(* IEC 61131-3 sources: std_i2980_v2.06_cp053/Source/IMM/ieccontrol/NozzleGeneral, 10 files *)

(* ---- ABButtonControl.pu ---- *)
IMPORT_OVER_LISTFILE
 IS_LINKED
, cBarInvert
, tyPanelButton
, tevPanelButtonRegisterData
, tevPanelButtonRegister
, ABManualButton
, tsDeviceId
, tsPanelButton

END_IMPORT

ALGORITHM_BLOCK ABButtonControl #DUMMY_EDIT_BLOCK

SYSTEM_VAR
 sv_bInitStart : BOOL;
 sv_bDeviceReady : BOOL;
 sv_bTransducerAvailable : BOOL;
 sv_iPanelMovementSelector : DINT;
 sv_PanelButtons : tyPanelButton;
 di_ButtonFwd : BOOL;
 di_ButtonBwd : BOOL;
 sv_bNozzleFwd : BOOL;
 sv_bNozzleBwd : BOOL;
 sv_bButtonFwd : BOOL;
 sv_bButtonBwd : BOOL;
 di_ButtonGeneral1 : BOOL;
 di_ButtonGeneral2 : BOOL;
 sv_DeviceId : tsDeviceId;
 sv_rNozzlePosition : REAL;
 sv_rNozzleStroke : REAL;
END_VAR

SYSTEM_OBJECT
 evPanelButtonRegister : tevPanelButtonRegister;
 PU_Task_7 : TASK;
 PU_Task_13 : TASK;
END_OBJECT

VAR
 evPanelButtonRegisterData : tevPanelButtonRegisterData;
 abManualButton : ABManualButton;
 mpbButtonGeneralFwd : REFTO BOOL;
 mpbButtonGeneralBwd : REFTO BOOL;
 mbDIButtonFwdLinked : BOOL;
 mbDIButtonBwdLinked : BOOL;
 mbDIButtonGeneralFwdLinked : BOOL;
 mbDIButtonGeneralBwdLinked : BOOL;
 mpiPanelMovementSelector : REFTO DINT;
END_VAR

VAR CONSTANT
 cButtonMoveFwdBwd : DINT := 1;
END_VAR

POSTUPDATE_ALGORITHM pRegisterButtons ON PU_Task_13 WITH sv_bInitStart

#BEGIN_EDIT_BLOCK
(**************************************** WARNING ********************************************
 *** The KEBA Kemro K2 System including software is not intended for safety control tasks! ***
 ***                       For further information see Comment tab!                        ***
 *********************************************************************************************)

mpbButtonGeneralFwd := EMPTY;
mpbButtonGeneralBwd := EMPTY;

mbDIButtonFwdLinked := IS_LINKED(di_ButtonFwd);
mbDIButtonBwdLinked := IS_LINKED(di_ButtonBwd);

mbDIButtonGeneralFwdLinked := IS_LINKED(di_ButtonGeneral1);
mbDIButtonGeneralBwdLinked := IS_LINKED(di_ButtonGeneral2);

IF (mbDIButtonGeneralFwdLinked AND mbDIButtonGeneralBwdLinked) THEN
    mpiPanelMovementSelector := @sv_iPanelMovementSelector;
END_IF;

evPanelButtonRegisterData.Button.nPanelButtonType := nPanelButtonMovement;
evPanelButtonRegisterData.Button.iCompId := sv_DeviceId.CompId;
evPanelButtonRegisterData.Button.iIndexId := sv_DeviceId.IndexId;
evPanelButtonRegisterData.Button.iButtonId := cButtonMoveFwdBwd;
evPanelButtonRegisterData.Button.pbActionVar1 := @sv_bButtonFwd;
evPanelButtonRegisterData.Button.pbActionVar2 := @sv_bButtonBwd;
IF sv_bTransducerAvailable THEN
   evPanelButtonRegisterData.Button.Optional.prActVar := @sv_rNozzlePosition;
END_IF;
evPanelButtonRegisterData.Button.Optional.prMaxVar := @sv_rNozzleStroke;
evPanelButtonRegisterData.Button.Optional.prMinVar :=  EMPTY;
evPanelButtonRegisterData.Button.Optional.iBarAttr := cBarInvert;
evPanelButtonRegisterData.Button.Optional.pbLimitSwitch1 := @sv_bNozzleFwd;
evPanelButtonRegisterData.Button.Optional.pbLimitSwitch2 := @sv_bNozzleBwd;
SET_EVENT(evPanelButtonRegister, evPanelButtonRegisterData);

;#END_EDIT_BLOCK END_ALGORITHM

POSTUPDATE_ALGORITHM pButtonFwd ON PU_Task_7 WITH di_ButtonFwd, sv_bButtonFwd, mpbButtonGeneralFwd^

VAR
 bButton : BOOL;
END_VAR
#BEGIN_EDIT_BLOCK
(**************************************** WARNING ********************************************
 *** The KEBA Kemro K2 System including software is not intended for safety control tasks! ***
 ***                       For further information see Comment tab!                        ***
 *********************************************************************************************)

// soft panel button
bButton := sv_bButtonFwd;

// hw panel button
IF mbDIButtonFwdLinked THEN
    bButton := bButton OR di_ButtonFwd;
END_IF;

// external panel button
IF CHECK_REF(mpbButtonGeneralFwd^) THEN
    bButton := bButton OR mpbButtonGeneralFwd^;
END_IF;

abManualButton.aButtonFwd(bButtonFwd := bButton);

;#END_EDIT_BLOCK END_ALGORITHM

POSTUPDATE_ALGORITHM pButtonBwd ON PU_Task_7 WITH di_ButtonBwd, sv_bButtonBwd, mpbButtonGeneralBwd^

VAR
 bButton : BOOL;
END_VAR
#BEGIN_EDIT_BLOCK
(**************************************** WARNING ********************************************
 *** The KEBA Kemro K2 System including software is not intended for safety control tasks! ***
 ***                       For further information see Comment tab!                        ***
 *********************************************************************************************)

// soft panel button
bButton := sv_bButtonBwd;

// hw panel button
IF mbDIButtonBwdLinked THEN
    bButton := bButton OR di_ButtonBwd;
END_IF;

// external panel button
IF CHECK_REF(mpbButtonGeneralBwd^) THEN
    bButton := bButton OR mpbButtonGeneralBwd^;
END_IF;

abManualButton.aButtonBwd(bButtonBwd := bButton);

;#END_EDIT_BLOCK END_ALGORITHM

POSTUPDATE_ALGORITHM pMoveSelectorChanged ON PU_Task_7 WITH mpiPanelMovementSelector^

VAR
 Button : tsPanelButton;
END_VAR
#BEGIN_EDIT_BLOCK
(**************************************** WARNING ********************************************
 *** The KEBA Kemro K2 System including software is not intended for safety control tasks! ***
 ***                       For further information see Comment tab!                        ***
 *********************************************************************************************)

mpbButtonGeneralFwd := EMPTY;
mpbButtonGeneralBwd := EMPTY;

IF (NOT sv_bDeviceReady) THEN
    // stop active movements
    abManualButton.aButtonBwd(bButtonBwd := FALSE);
    abManualButton.aButtonFwd(bButtonFwd := FALSE);
END_IF;

IF (sv_iPanelMovementSelector > 0) THEN
    Button := sv_PanelButtons[sv_iPanelMovementSelector];
    IF Button.iCompId = sv_DeviceId.CompId AND
        Button.iIndexId = sv_DeviceId.IndexId THEN
        IF Button.iButtonId = cButtonMoveFwdBwd THEN
            mpbButtonGeneralFwd := @di_ButtonGeneral1;
            mpbButtonGeneralBwd := @di_ButtonGeneral2;
        END_IF;
    END_IF;
END_IF;

;#END_EDIT_BLOCK END_ALGORITHM

END_ALGORITHM_BLOCK

#END_OF_IEC_PART

@Puma @IecEditor 6 150 @Pou 25
@@@BEG_Comment@@@

@@@END_Comment@@@

@BEG_Contents

@BEG_Func
@RT(17)FuncTreeContainer
1
@Var @RT(9)IS_LINKED @RT(0) @T @T @DERIVED 0 @F @RT(22)KEBA_STANDARD_FUNCTION @F
@T
@BEG_Attrib
0 @RT(0) @RT(0)
@END_Attrib
1 1 @F @F @F @F

@END_Func

@BEG_Const
@RT(18)ConstTreeContainer
1
@Var @RT(10)cBarInvert @RT(0) @T @F @DT @RT(4)BYTE @RT(0) @T @T @BASIC 0 @F
@F @F
@T
@BEG_Attrib
0 @RT(1)1 @RT(0)
@END_Attrib
1 1 @F @F @F @F

@END_Const

@BEG_Export

@BEG_Kind
@ALGORITHM_BLOCK @RT(15)ABButtonControl @STRUCTURED_TEXT
@RT(0) @RT(0) @RT(0)
@END_Kind

@BEG_Dcl
@RT(16)DclTreeContainer
29
@Var @RT(13)sv_bInitStart @RT(0) @T @T @RENAMED 0 @T @T @DT @RT(4)BOOL @RT(0) @T @T @BASIC 0 @F
@F @F
@T
@BEG_Attrib
3 @RT(0) @RT(0) @RT(0)
@END_Attrib
1 8 @F @F @F @F

@Var @RT(15)sv_bDeviceReady @RT(0) @T @T @RENAMED 0 @T @T @DT @RT(4)BOOL @RT(0) @T @T @BASIC 0 @F
@F @F
@T
@BEG_Attrib
3 @RT(0) @RT(0) @RT(0)
@END_Attrib
1 8 @F @F @F @F

@Var @RT(23)sv_bTransducerAvailable @RT(0) @T @F @DT @RT(4)BOOL @RT(0) @T @T @BASIC 0 @F
@F @F
@T
@BEG_Attrib
3 @RT(0) @RT(0) @RT(0)
@END_Attrib
1 8 @F @F @F @F

@Var @RT(25)sv_iPanelMovementSelector @RT(0) @T @F @DT @RT(4)DINT @RT(0) @T @T @BASIC 0 @F
@F @F
@T
@BEG_Attrib
3 @RT(0) @RT(0) @RT(0)
@END_Attrib
1 8 @F @F @F @F

@Var @RT(15)sv_PanelButtons @RT(0) @T @T @DERIVED 0 @T @T @DT @RT(13)tyPanelButton @RT(0) @T @T @UNKNOWN 0 @F
@F @F
@T
@BEG_Attrib
3 @RT(0) @RT(0) @RT(0)
@END_Attrib
1 8 @F @F @F @F

@Var @RT(25)evPanelButtonRegisterData @RT(0) @T @T @DERIVED 0 @T @T @DT @RT(26)tevPanelButtonRegisterData @RT(0) @T @T @UNKNOWN 0 @F
@F @F
@T
@BEG_Attrib
3 @RT(0) @RT(0) @RT(0)
@END_Attrib
1 0 @F @F @F @F

@Var @RT(21)evPanelButtonRegister @RT(0) @T @T @DERIVED 0 @T @T @DT @RT(22)tevPanelButtonRegister @RT(0) @T @T @UNKNOWN 0 @F
@F @F
@T
@BEG_Attrib
3 @RT(0) @RT(0) @RT(0)
@END_Attrib
1 7 @F @F @F @F

@Var @RT(14)abManualButton @RT(0) @T @T @DERIVED 0 @T @T @DT @RT(14)ABManualButton @RT(0) @T @T @UNKNOWN 0 @F
@F @F
@T
@BEG_Attrib
3 @RT(0) @RT(0) @RT(0)
@END_Attrib
1 0 @F @F @F @F

@Var @RT(12)di_ButtonFwd @RT(0) @T @T @RENAMED 0 @T @T @DT @RT(4)BOOL @RT(0) @T @T @BASIC 0 @F
@F @F
@T
@BEG_Attrib
3 @RT(0) @RT(0) @RT(0)
@END_Attrib
1 8 @F @F @F @F

@Var @RT(12)di_ButtonBwd @RT(0) @T @T @RENAMED 0 @T @T @DT @RT(4)BOOL @RT(0) @T @T @BASIC 0 @F
@F @F
@T
@BEG_Attrib
3 @RT(0) @RT(0) @RT(0)
@END_Attrib
1 8 @F @F @F @F

@Var @RT(13)sv_bNozzleFwd @RT(0) @T @T @RENAMED 0 @T @T @DT @RT(4)BOOL @RT(0) @T @T @BASIC 0 @F
@F @F
@T
@BEG_Attrib
3 @RT(0) @RT(0) @RT(0)
@END_Attrib
1 8 @F @F @F @F

@Var @RT(13)sv_bNozzleBwd @RT(0) @T @T @RENAMED 0 @T @T @DT @RT(4)BOOL @RT(0) @T @T @BASIC 0 @F
@F @F
@T
@BEG_Attrib
3 @RT(0) @RT(0) @RT(0)
@END_Attrib
1 8 @F @F @F @F

@Var @RT(13)sv_bButtonFwd @RT(0) @T @T @RENAMED 0 @T @T @DT @RT(4)BOOL @RT(0) @T @T @BASIC 0 @F
@F @F
@T
@BEG_Attrib
3 @RT(0) @RT(0) @RT(0)
@END_Attrib
1 8 @F @F @F @F

@Var @RT(13)sv_bButtonBwd @RT(0) @T @T @RENAMED 0 @T @T @DT @RT(4)BOOL @RT(0) @T @T @BASIC 0 @F
@F @F
@T
@BEG_Attrib
3 @RT(0) @RT(0) @RT(0)
@END_Attrib
1 8 @F @F @F @F

@Var @RT(17)di_ButtonGeneral1 @RT(0) @T @F @DT @RT(4)BOOL @RT(0) @T @T @BASIC 0 @F
@F @F
@T
@BEG_Attrib
3 @RT(0) @RT(0) @RT(0)
@END_Attrib
1 8 @F @F @F @F

@Var @RT(17)di_ButtonGeneral2 @RT(0) @T @F @DT @RT(4)BOOL @RT(0) @T @T @BASIC 0 @F
@F @F
@T
@BEG_Attrib
3 @RT(0) @RT(0) @RT(0)
@END_Attrib
1 8 @F @F @F @F

@Var @RT(9)PU_Task_7 @RT(0) @T @F @DT @RT(4)TASK @RT(0) @T @T @BASIC 0 @F
@F @F
@T
@BEG_Attrib
3 @RT(0) @RT(0) @RT(0)
@END_Attrib
1 7 @F @F @F @F

@Var @RT(10)PU_Task_13 @RT(0) @T @T @RENAMED 0 @T @T @DT @RT(4)TASK @RT(0) @T @T @BASIC 0 @F
@F @F
@T
@BEG_Attrib
3 @RT(0) @RT(0) @RT(0)
@END_Attrib
1 7 @F @F @F @F

@Var @RT(11)sv_DeviceId @RT(0) @T @T @DERIVED 0 @T @T @DT @RT(10)tsDeviceId @RT(0) @T @T @UNKNOWN 0 @F
@F @F
@T
@BEG_Attrib
3 @RT(0) @RT(0) @RT(0)
@END_Attrib
1 8 @F @F @F @F

@Var @RT(18)sv_rNozzlePosition @RT(0) @T @F @DT @RT(4)REAL @RT(0) @T @T @BASIC 0 @F
@F @F
@T
@BEG_Attrib
3 @RT(0) @RT(0) @RT(0)
@END_Attrib
1 8 @F @F @F @F

@Var @RT(16)sv_rNozzleStroke @RT(0) @T @F @DT @RT(4)REAL @RT(0) @T @T @BASIC 0 @F
@F @F
@T
@BEG_Attrib
3 @RT(0) @RT(0) @RT(0)
@END_Attrib
1 8 @F @F @F @F

@Var @RT(17)cButtonMoveFwdBwd @RT(0) @T @F @DT @RT(4)DINT @RT(0) @T @T @BASIC 0 @F
@F @F
@T
@BEG_Attrib
3 @RT(1)1 @RT(0) @RT(0)
@END_Attrib
1 15 @F @F @F @F

@Var @RT(19)mpbButtonGeneralFwd @RT(0) @T @T @REFTO 0 @T @DT @RT(4)BOOL @RT(0) @T @T @BASIC 0 @F
@F @F
@T
@BEG_Attrib
3 @RT(0) @RT(0) @RT(0)
@END_Attrib
1 0 @F @F @F @F

@Var @RT(19)mpbButtonGeneralBwd @RT(0) @T @T @REFTO 0 @T @DT @RT(4)BOOL @RT(0) @T @T @BASIC 0 @F
@F @F
@T
@BEG_Attrib
3 @RT(0) @RT(0) @RT(0)
@END_Attrib
1 0 @F @F @F @F

@Var @RT(19)mbDIButtonFwdLinked @RT(0) @T @F @DT @RT(4)BOOL @RT(0) @T @T @BASIC 0 @F
@F @F
@T
@BEG_Attrib
3 @RT(0) @RT(0) @RT(0)
@END_Attrib
1 0 @F @F @F @F

@Var @RT(19)mbDIButtonBwdLinked @RT(0) @T @F @DT @RT(4)BOOL @RT(0) @T @T @BASIC 0 @F
@F @F
@T
@BEG_Attrib
3 @RT(0) @RT(0) @RT(0)
@END_Attrib
1 0 @F @F @F @F

@Var @RT(26)mbDIButtonGeneralFwdLinked @RT(0) @T @F @DT @RT(4)BOOL @RT(0) @T @T @BASIC 0 @F
@F @F
@T
@BEG_Attrib
3 @RT(0) @RT(0) @RT(0)
@END_Attrib
1 0 @F @F @F @F

@Var @RT(26)mbDIButtonGeneralBwdLinked @RT(0) @T @F @DT @RT(4)BOOL @RT(0) @T @T @BASIC 0 @F
@F @F
@T
@BEG_Attrib
3 @RT(0) @RT(0) @RT(0)
@END_Attrib
1 0 @F @F @F @F

@Var @RT(24)mpiPanelMovementSelector @RT(0) @T @T @REFTO 0 @T @DT @RT(4)DINT @RT(0) @T @T @BASIC 0 @F
@F @F
@T
@BEG_Attrib
3 @RT(0) @RT(0) @RT(0)
@END_Attrib
1 0 @F @F @F @F

@END_Dcl

@END_Export

@BEG_Body

4

@BEG_Export

@BEG_Algo
@POSTUPDATE_ALGORITHM @RT(16)pRegisterButtons @STRUCTURED_TEXT
@RT(0) @RT(13)sv_bInitStart @RT(10)PU_Task_13 @F @F
@END_Algo

@BEG_Dcl
@RT(16)DclTreeContainer
0
@END_Dcl

@END_Export

@BEG_Export

@BEG_Algo
@POSTUPDATE_ALGORITHM @RT(10)pButtonFwd @STRUCTURED_TEXT
@RT(0) @RT(49)di_ButtonFwd, sv_bButtonFwd, mpbButtonGeneralFwd^ @RT(9)PU_Task_7 @F @F
@END_Algo

@BEG_Dcl
@RT(16)DclTreeContainer
1
@Var @RT(7)bButton @RT(0) @T @F @DT @RT(4)BOOL @RT(0) @T @T @BASIC 0 @F
@F @F
@T
@BEG_Attrib
3 @RT(0) @RT(0) @RT(0)
@END_Attrib
1 0 @F @F @F @F

@END_Dcl

@END_Export

@BEG_Export

@BEG_Algo
@POSTUPDATE_ALGORITHM @RT(10)pButtonBwd @STRUCTURED_TEXT
@RT(0) @RT(49)di_ButtonBwd, sv_bButtonBwd, mpbButtonGeneralBwd^ @RT(9)PU_Task_7 @F @F
@END_Algo

@BEG_Dcl
@RT(16)DclTreeContainer
1
@Var @RT(7)bButton @RT(0) @T @F @DT @RT(4)BOOL @RT(0) @T @T @BASIC 0 @F
@F @F
@T
@BEG_Attrib
3 @RT(0) @RT(0) @RT(0)
@END_Attrib
1 0 @F @F @F @F

@END_Dcl

@END_Export

@BEG_Export

@BEG_Algo
@POSTUPDATE_ALGORITHM @RT(20)pMoveSelectorChanged @STRUCTURED_TEXT
@RT(0) @RT(25)mpiPanelMovementSelector^ @RT(9)PU_Task_7 @F @F
@END_Algo

@BEG_Dcl
@RT(16)DclTreeContainer
1
@Var @RT(6)Button @RT(0) @T @T @DERIVED 0 @T @T @DT @RT(13)tsPanelButton @RT(0) @T @T @UNKNOWN 0 @F
@F @F
@T
@BEG_Attrib
3 @RT(0) @RT(0) @RT(0)
@END_Attrib
1 0 @F @F @F @F

@END_Dcl

@END_Export

@BEG_Body
@TL(35)
(**************************************** WARNING ********************************************
 *** The KEBA Kemro K2 System including software is not intended for safety control tasks! ***
 ***                       For further information see Comment tab!                        ***
 *********************************************************************************************)

mpbButtonGeneralFwd := EMPTY;
mpbButtonGeneralBwd := EMPTY;

mbDIButtonFwdLinked := IS_LINKED(di_ButtonFwd);
mbDIButtonBwdLinked := IS_LINKED(di_ButtonBwd);

mbDIButtonGeneralFwdLinked := IS_LINKED(di_ButtonGeneral1);
mbDIButtonGeneralBwdLinked := IS_LINKED(di_ButtonGeneral2);

IF (mbDIButtonGeneralFwdLinked AND mbDIButtonGeneralBwdLinked) THEN
    mpiPanelMovementSelector := @sv_iPanelMovementSelector;
END_IF;

evPanelButtonRegisterData.Button.nPanelButtonType := nPanelButtonMovement;
evPanelButtonRegisterData.Button.iCompId := sv_DeviceId.CompId;
evPanelButtonRegisterData.Button.iIndexId := sv_DeviceId.IndexId;
evPanelButtonRegisterData.Button.iButtonId := cButtonMoveFwdBwd;
evPanelButtonRegisterData.Button.pbActionVar1 := @sv_bButtonFwd;
evPanelButtonRegisterData.Button.pbActionVar2 := @sv_bButtonBwd;
IF sv_bTransducerAvailable THEN
   evPanelButtonRegisterData.Button.Optional.prActVar := @sv_rNozzlePosition;
END_IF;
evPanelButtonRegisterData.Button.Optional.prMaxVar := @sv_rNozzleStroke;
evPanelButtonRegisterData.Button.Optional.prMinVar :=  EMPTY;
evPanelButtonRegisterData.Button.Optional.iBarAttr := cBarInvert;
evPanelButtonRegisterData.Button.Optional.pbLimitSwitch1 := @sv_bNozzleFwd;
evPanelButtonRegisterData.Button.Optional.pbLimitSwitch2 := @sv_bNozzleBwd;
SET_EVENT(evPanelButtonRegister, evPanelButtonRegisterData);

@END_Body

@@@BEG_Comment@@@
@TL(0)

@@@END_Comment@@@

@BEG_Body
@TL(21)
(**************************************** WARNING ********************************************
 *** The KEBA Kemro K2 System including software is not intended for safety control tasks! ***
 ***                       For further information see Comment tab!                        ***
 *********************************************************************************************)

// soft panel button
bButton := sv_bButtonFwd;

// hw panel button
IF mbDIButtonFwdLinked THEN
    bButton := bButton OR di_ButtonFwd;
END_IF;

// external panel button
IF CHECK_REF(mpbButtonGeneralFwd^) THEN
    bButton := bButton OR mpbButtonGeneralFwd^;
END_IF;

abManualButton.aButtonFwd(bButtonFwd := bButton);

@END_Body

@@@BEG_Comment@@@
@TL(0)

@@@END_Comment@@@

@BEG_Body
@TL(20)
(**************************************** WARNING ********************************************
 *** The KEBA Kemro K2 System including software is not intended for safety control tasks! ***
 ***                       For further information see Comment tab!                        ***
 *********************************************************************************************)

// soft panel button
bButton := sv_bButtonBwd;

// hw panel button
IF mbDIButtonBwdLinked THEN
    bButton := bButton OR di_ButtonBwd;
END_IF;

// external panel button
IF CHECK_REF(mpbButtonGeneralBwd^) THEN
    bButton := bButton OR mpbButtonGeneralBwd^;
END_IF;

abManualButton.aButtonBwd(bButtonBwd := bButton);

@END_Body

@@@BEG_Comment@@@
@TL(0)

@@@END_Comment@@@

@BEG_Body
@TL(27)
(**************************************** WARNING ********************************************
 *** The KEBA Kemro K2 System including software is not intended for safety control tasks! ***
 ***                       For further information see Comment tab!                        ***
 *********************************************************************************************)

mpbButtonGeneralFwd := EMPTY;
mpbButtonGeneralBwd := EMPTY;

IF (NOT sv_bDeviceReady) THEN
    // stop active movements
    abManualButton.aButtonBwd(bButtonBwd := FALSE);
    abManualButton.aButtonFwd(bButtonFwd := FALSE);
END_IF;

IF (sv_iPanelMovementSelector > 0) THEN
    Button := sv_PanelButtons[sv_iPanelMovementSelector];
    IF Button.iCompId = sv_DeviceId.CompId AND
        Button.iIndexId = sv_DeviceId.IndexId THEN
        IF Button.iButtonId = cButtonMoveFwdBwd THEN
            mpbButtonGeneralFwd := @di_ButtonGeneral1;
            mpbButtonGeneralBwd := @di_ButtonGeneral2;
        END_IF;
    END_IF;
END_IF;

@END_Body

@@@BEG_Comment@@@
@TL(0)

@@@END_Comment@@@
@END_Body

@END_Contents

(* ---- ABChangeProfile.pu ---- *)
IMPORT_OVER_LISTFILE
 KAPPL_VisProfile
, tnDataState
, FBChangeNoOfProfileSteps

END_IMPORT

ALGORITHM_BLOCK ABChangeProfile #DUMMY_EDIT_BLOCK

SYSTEM_VAR
 sv_NozzleBwdProfVis : KAPPL_VisProfile;
 sv_bUseStartPosProfiles : BOOL;
 sv_bInitStart : BOOL;
 sv_NozzleFwdProfVis : KAPPL_VisProfile;
 sv_DataState : tnDataState;
END_VAR

SYSTEM_OBJECT
 PU_Task_7 : TASK;
END_OBJECT

POSTUPDATE_ALGORITHM pChangeBwdProfile ON PU_Task_7 WITH sv_NozzleBwdProfVis, sv_bInitStart

VAR
 fbChangeNoOfProfileStepsBwd : FBChangeNoOfProfileSteps;
END_VAR
#BEGIN_EDIT_BLOCK
fbChangeNoOfProfileStepsBwd(ProfileVis := sv_NozzleBwdProfVis.Profile,
                            bUseStartPosProfiles := sv_bUseStartPosProfiles,
                            bOpenEndProfile := sv_NozzleBwdProfVis.bOpenEndProfile,
                            bDataStateIsReady := (sv_DataState = nReady));

;#END_EDIT_BLOCK END_ALGORITHM

POSTUPDATE_ALGORITHM pChangeFwdProfile ON PU_Task_7 WITH sv_NozzleFwdProfVis, sv_bInitStart

VAR
 fbChangeNoOfProfileStepsFwd : FBChangeNoOfProfileSteps;
END_VAR
#BEGIN_EDIT_BLOCK
fbChangeNoOfProfileStepsFwd(ProfileVis := sv_NozzleFwdProfVis.Profile,
                            bUseStartPosProfiles := sv_bUseStartPosProfiles,
                            bOpenEndProfile := sv_NozzleFwdProfVis.bOpenEndProfile,
                            bDataStateIsReady := (sv_DataState = nReady));

;#END_EDIT_BLOCK END_ALGORITHM

END_ALGORITHM_BLOCK

#END_OF_IEC_PART

@Puma @IecEditor 6 103 @Pou 25
@@@BEG_Comment@@@

@@@END_Comment@@@

@BEG_Contents

@BEG_Func
@RT(17)FuncTreeContainer
0
@END_Func

@BEG_Const
@RT(18)ConstTreeContainer
0
@END_Const

@BEG_Export

@BEG_Kind
@ALGORITHM_BLOCK @RT(15)ABChangeProfile @STRUCTURED_TEXT
@RT(0) @RT(0) @RT(0)
@END_Kind

@BEG_Dcl
@RT(16)DclTreeContainer
6
@Var @RT(9)PU_Task_7 @RT(0) @T @T @RENAMED 0 @T @T @DT @RT(4)TASK @RT(0) @T @T @BASIC 0 @F
@F @F
@T
@BEG_Attrib
3 @RT(0) @RT(0) @RT(0)
@END_Attrib
1 7 @F @F @F @F

@Var @RT(19)sv_NozzleBwdProfVis @RT(0) @T @T @DERIVED 0 @T @T @DT @RT(16)KAPPL_VisProfile @RT(0) @T @T @UNKNOWN 0 @F
@F @F
@T
@BEG_Attrib
3 @RT(0) @RT(0) @RT(0)
@END_Attrib
1 8 @F @F @F @F

@Var @RT(23)sv_bUseStartPosProfiles @RT(0) @T @F @DT @RT(4)BOOL @RT(0) @T @T @BASIC 0 @F
@F @F
@T
@BEG_Attrib
3 @RT(0) @RT(0) @RT(0)
@END_Attrib
1 8 @F @F @F @F

@Var @RT(13)sv_bInitStart @RT(0) @T @F @DT @RT(4)BOOL @RT(0) @T @T @BASIC 0 @F
@F @F
@T
@BEG_Attrib
3 @RT(0) @RT(0) @RT(0)
@END_Attrib
1 8 @F @F @F @F

@Var @RT(19)sv_NozzleFwdProfVis @RT(0) @T @T @RENAMED 0 @T @T @DT @RT(16)KAPPL_VisProfile @RT(0) @T @T @UNKNOWN 0 @F
@F @F
@T
@BEG_Attrib
3 @RT(0) @RT(0) @RT(0)
@END_Attrib
1 8 @F @F @F @F

@Var @RT(12)sv_DataState @RT(0) @T @T @DERIVED 0 @T @T @DT @RT(11)tnDataState @RT(0) @T @T @UNKNOWN 0 @F
@F @F
@T
@BEG_Attrib
3 @RT(0) @RT(0) @RT(0)
@END_Attrib
1 8 @F @F @F @F

@END_Dcl

@END_Export

@BEG_Body

2

@BEG_Export

@BEG_Algo
@POSTUPDATE_ALGORITHM @RT(17)pChangeBwdProfile @STRUCTURED_TEXT
@RT(0) @RT(34)sv_NozzleBwdProfVis, sv_bInitStart @RT(9)PU_Task_7 @F @F
@END_Algo

@BEG_Dcl
@RT(16)DclTreeContainer
1
@Var @RT(27)fbChangeNoOfProfileStepsBwd @RT(0) @T @T @DERIVED 0 @T @T @DT @RT(24)FBChangeNoOfProfileSteps @RT(0) @T @T @UNKNOWN 0 @F
@F @F
@T
@BEG_Attrib
3 @RT(0) @RT(0) @RT(0)
@END_Attrib
1 0 @F @F @F @F

@END_Dcl

@END_Export

@BEG_Export

@BEG_Algo
@POSTUPDATE_ALGORITHM @RT(17)pChangeFwdProfile @STRUCTURED_TEXT
@RT(0) @RT(34)sv_NozzleFwdProfVis, sv_bInitStart @RT(9)PU_Task_7 @F @F
@END_Algo

@BEG_Dcl
@RT(16)DclTreeContainer
1
@Var @RT(27)fbChangeNoOfProfileStepsFwd @RT(0) @T @T @DERIVED 0 @T @T @DT @RT(24)FBChangeNoOfProfileSteps @RT(0) @T @T @UNKNOWN 0 @F
@F @F
@T
@BEG_Attrib
3 @RT(0) @RT(0) @RT(0)
@END_Attrib
1 0 @F @F @F @F

@END_Dcl

@END_Export

@BEG_Body
@TL(6)
fbChangeNoOfProfileStepsBwd(ProfileVis := sv_NozzleBwdProfVis.Profile,
                            bUseStartPosProfiles := sv_bUseStartPosProfiles,
                            bOpenEndProfile := sv_NozzleBwdProfVis.bOpenEndProfile,
                            bDataStateIsReady := (sv_DataState = nReady));

@END_Body

@@@BEG_Comment@@@
@TL(0)

@@@END_Comment@@@

@BEG_Body
@TL(6)
fbChangeNoOfProfileStepsFwd(ProfileVis := sv_NozzleFwdProfVis.Profile,
                            bUseStartPosProfiles := sv_bUseStartPosProfiles,
                            bOpenEndProfile := sv_NozzleFwdProfVis.bOpenEndProfile,
                            bDataStateIsReady := (sv_DataState = nReady));

@END_Body

@@@BEG_Comment@@@
@TL(0)

@@@END_Comment@@@
@END_Body

@END_Contents

(* ---- ABCheckNozzleFwd.pu ---- *)
(*
@h    ! WARNING !
@h    The Kemro K2 system (including software) only meets category B according to EN 954-1,
@h    thus it is not intended for usage in safety-relevant control applications in the field
@h    of personal safety (e.g. emergency stop).
@h    To implement potentially necessary safety-relevant control tasks, always use additional
@h    external safety devices that are intended for the particular purpose, and meet the necessary
@h    functional safety.
@h    For further information see EN 954-1 (EN ISO 13849-1) and/or the K2-x00 user manual, chapter
@h    "CE conformity, directives and standards".

This block locks all movements of lockgroup cLockGroupNozzleFwd
with an according alarm if the nozzle is in fwd position (sv_bNozzleFwd = TRUE)
*)

IMPORT_OVER_LISTFILE
 cCompOperationMode
, cModeAutomatic
, tsDeviceId
, FBLockUnlockGroup

END_IMPORT

ALGORITHM_BLOCK ABCheckNozzleFwd #DUMMY_EDIT_BLOCK

SYSTEM_VAR
 sv_bInitDone : BOOL;
 sv_bNozzleFwd : BOOL;
 sv_DeviceId : tsDeviceId;
END_VAR

SYSTEM_OBJECT
 PU_Task_7 : TASK;
 erNozzleMustNotBeFwd : ALARM;
END_OBJECT

POSTUPDATE_ALGORITHM pNozzleFwd ON PU_Task_7 WITH sv_bNozzleFwd,sv_bInitDone

VAR
 fbLockUnlockGroup : FBLockUnlockGroup;
 bInitDone : BOOL;
END_VAR
#BEGIN_EDIT_BLOCK
(**************************************** WARNING ********************************************
 *** The KEBA Kemro K2 System including software is not intended for safety control tasks! ***
 ***                       For further information see Comment tab!                        ***
 *********************************************************************************************)

IF NOT sv_bInitDone THEN
   RETURN;     // do not allow lock/unlock bevor init done
END_IF;

IF NOT bInitDone THEN
   fbLockUnlockGroup.Alarm.AlarmId :=erNozzleMustNotBeFwd;
   fbLockUnlockGroup.Alarm.SubId[1] := sv_DeviceId.CompId;
   fbLockUnlockGroup.Alarm.SubId[2] := sv_DeviceId.IndexId;
   fbLockUnlockGroup.Group := cLockGroupNozzleFwd;
   bInitDone := TRUE;
END_IF;

IF sv_bNozzleFwd THEN
   // nozzle fwd -> don't allow MoldHeightAdjust(Auto)
   fbLockUnlockGroup.Mode := nLockAbort;
ELSE
   // nozzle NOT fwd -> allow MoldHeightAdjust(Auto)
   fbLockUnlockGroup.Mode := nUnlock;
END_IF;

fbLockUnlockGroup();

;#END_EDIT_BLOCK END_ALGORITHM

END_ALGORITHM_BLOCK

#END_OF_IEC_PART

@Puma @IecEditor 6 97 @Pou 25
@@@BEG_Comment@@@
@h    ! WARNING !
@h    The Kemro K2 system (including software) only meets category B according to EN 954-1,
@h    thus it is not intended for usage in safety-relevant control applications in the field
@h    of personal safety (e.g. emergency stop).
@h    To implement potentially necessary safety-relevant control tasks, always use additional
@h    external safety devices that are intended for the particular purpose, and meet the necessary
@h    functional safety.
@h    For further information see EN 954-1 (EN ISO 13849-1) and/or the K2-x00 user manual, chapter
@h    "CE conformity, directives and standards".

This block locks all movements of lockgroup cLockGroupNozzleFwd
with an according alarm if the nozzle is in fwd position (sv_bNozzleFwd = TRUE)
@@@END_Comment@@@

@BEG_Contents

@BEG_Func
@RT(17)FuncTreeContainer
0
@END_Func

@BEG_Const
@RT(18)ConstTreeContainer
2
@Var @RT(18)cCompOperationMode @RT(0) @T @F @DT @RT(4)DINT @RT(0) @T @T @BASIC 0 @F
@F @F
@T
@BEG_Attrib
0 @RT(3)111 @RT(24)Component Operation Mode
@END_Attrib
1 1 @F @F @F @F

@Var @RT(14)cModeAutomatic @RT(0) @T @F @DT @RT(4)DINT @RT(0) @T @T @BASIC 0 @F
@F @F
@T
@BEG_Attrib
0 @RT(2)23 @RT(50)for locking/unlocking half and full automatic mode
@END_Attrib
1 1 @F @F @F @F

@END_Const

@BEG_Export

@BEG_Kind
@ALGORITHM_BLOCK @RT(16)ABCheckNozzleFwd @STRUCTURED_TEXT
@RT(0) @RT(0) @RT(0)
@END_Kind

@BEG_Dcl
@RT(16)DclTreeContainer
5
@Var @RT(9)PU_Task_7 @RT(0) @T @T @RENAMED 0 @T @T @DT @RT(4)TASK @RT(0) @T @T @BASIC 0 @F
@F @F
@T
@BEG_Attrib
3 @RT(0) @RT(0) @RT(0)
@END_Attrib
1 7 @F @F @F @F

@Var @RT(12)sv_bInitDone @RT(0) @T @F @DT @RT(4)BOOL @RT(0) @T @T @BASIC 0 @F
@F @F
@T
@BEG_Attrib
3 @RT(0) @RT(0) @RT(0)
@END_Attrib
1 8 @F @F @F @F

@Var @RT(13)sv_bNozzleFwd @RT(0) @T @T @RENAMED 0 @T @T @DT @RT(4)BOOL @RT(0) @T @T @BASIC 0 @F
@F @F
@T
@BEG_Attrib
3 @RT(0) @RT(0) @RT(0)
@END_Attrib
1 8 @F @F @F @F

@Var @RT(20)erNozzleMustNotBeFwd @RT(0) @T @F @DT @RT(5)ALARM @RT(0) @T @T @BASIC 0 @F
@F @F
@T
@BEG_Attrib
3 @RT(0) @RT(0) @RT(0)
@END_Attrib
1 7 @F @F @F @F

@Var @RT(11)sv_DeviceId @RT(0) @T @T @DERIVED 0 @F @RT(10)tsDeviceId @F
@T
@BEG_Attrib
3 @RT(0) @RT(0) @RT(0)
@END_Attrib
1 8 @F @F @F @F

@END_Dcl

@END_Export

@BEG_Body

1

@BEG_Export

@BEG_Algo
@POSTUPDATE_ALGORITHM @RT(10)pNozzleFwd @STRUCTURED_TEXT
@RT(0) @RT(26)sv_bNozzleFwd,sv_bInitDone @RT(9)PU_Task_7 @F @F
@END_Algo

@BEG_Dcl
@RT(16)DclTreeContainer
2
@Var @RT(17)fbLockUnlockGroup @RT(0) @T @T @DERIVED 0 @F @RT(17)FBLockUnlockGroup @F
@T
@BEG_Attrib
3 @RT(0) @RT(0) @RT(0)
@END_Attrib
1 0 @F @F @F @F

@Var @RT(9)bInitDone @RT(0) @T @F @DT @RT(4)BOOL @RT(0) @T @T @BASIC 0 @F
@F @F
@T
@BEG_Attrib
3 @RT(0) @RT(0) @RT(0)
@END_Attrib
1 0 @F @F @F @F

@END_Dcl

@END_Export

@BEG_Body
@TL(28)
(**************************************** WARNING ********************************************
 *** The KEBA Kemro K2 System including software is not intended for safety control tasks! ***
 ***                       For further information see Comment tab!                        ***
 *********************************************************************************************)

IF NOT sv_bInitDone THEN
   RETURN;     // do not allow lock/unlock bevor init done
END_IF;

IF NOT bInitDone THEN
   fbLockUnlockGroup.Alarm.AlarmId :=erNozzleMustNotBeFwd;
   fbLockUnlockGroup.Alarm.SubId[1] := sv_DeviceId.CompId;
   fbLockUnlockGroup.Alarm.SubId[2] := sv_DeviceId.IndexId;
   fbLockUnlockGroup.Group := cLockGroupNozzleFwd;
   bInitDone := TRUE;
END_IF;

IF sv_bNozzleFwd THEN
   // nozzle fwd -> don't allow MoldHeightAdjust(Auto)
   fbLockUnlockGroup.Mode := nLockAbort;
ELSE
   // nozzle NOT fwd -> allow MoldHeightAdjust(Auto)
   fbLockUnlockGroup.Mode := nUnlock;
END_IF;

fbLockUnlockGroup();

@END_Body

@@@BEG_Comment@@@
@TL(0)

@@@END_Comment@@@
@END_Body

@END_Contents

(* ---- ABCheckSettings.pu ---- *)
(*
@h    ! WARNING !
@h    The Kemro K2 system (including software) only meets category B according to EN 954-1,
@h    thus it is not intended for usage in safety-relevant control applications in the field
@h    of personal safety (e.g. emergency stop).
@h    To implement potentially necessary safety-relevant control tasks, always use additional
@h    external safety devices that are intended for the particular purpose, and meet the necessary
@h    functional safety.
@h    For further information see EN 954-1 (EN ISO 13849-1) and/or the K2-x00 user manual, chapter
@h    "CE conformity, directives and standards".

AB set the refernces for the endposition monitor blocks.
This refernces denpend on the selected movement mode (position, limit or time)
In time mode the endposition monitoring is also done by this block.
*)

IMPORT_OVER_LISTFILE
 SET_ALARM
, START_PROCESS_ALGORITHM
, STOP_PROCESS_ALGORITHM
, nPositionDependent
, nMoveTimeDependent
, tnMovementMode
, tsEndPosData
, KAPPL_VisProfile
, tnNozzleMovementMode

END_IMPORT

ALGORITHM_BLOCK ABCheckSettings #DUMMY_EDIT_BLOCK

SYSTEM_VAR
 ai_Position : REAL;
 sv_MovementMode : tnMovementMode (* Nozzle Movement with Limitswitch or with position measurement *);
 sv_bInitStart : BOOL;
 sv_NozzleFwdMonData : tsEndPosData;
 sv_NozzleBwdMonData : tsEndPosData;
 di_LimitSwitchFwd : BOOL;
 di_LimitSwitchFwd2 : BOOL;
 sv_NozzleFwdProfVis : KAPPL_VisProfile;
 sv_NozzleBwdProfVis : KAPPL_VisProfile;
 di_LimitSwitchBwd : BOOL;
 sv_bNozzleFwd : BOOL;
 sv_bNozzleBwd : BOOL;
 sv_bFwdTimeReached : BOOL (* nozzle fwd time reached (for time dependent nozzle control) (must be FastRetain: cyclical change in AutoCycle) *);
 sv_bBwdTimeReached : BOOL (* nozzle bwd time reached (for time dependent nozzle control) (must be FastRetain: cyclical change in AutoCycle) *);
 sv_NozzleMovementMode : tnNozzleMovementMode;
END_VAR

SYSTEM_OBJECT
 PU_Task_3 : TASK;
END_OBJECT

POSTUPDATE_ALGORITHM pModeChanged ON PU_Task_3 WITH sv_MovementMode,sv_bInitStart

VAR_TEMP
 tmpFwd : tsEndPosData;
 tmpBwd : tsEndPosData;
END_VAR
#BEGIN_EDIT_BLOCK
(**************************************** WARNING ********************************************
 *** The KEBA Kemro K2 System including software is not intended for safety control tasks! ***
 ***                       For further information see Comment tab!                        ***
 *********************************************************************************************)

// update endposmon data when movement mode changes
// executed in PU_Task_3 so it is called before ABEndposMon.pParameterChanged

tmpFwd := sv_NozzleFwdMonData;
tmpBwd := sv_NozzleBwdMonData;

IF sv_MovementMode = nPositionDependent THEN
   //position depending
   tmpBwd.pbDI := EMPTY;
   tmpFwd.pbDI := EMPTY;
   tmpBwd.pProfile := @sv_NozzleBwdProfVis;
   tmpFwd.pProfile := @sv_NozzleFwdProfVis;

ELSIF sv_MovementMode = nLimitSwitchDependent THEN
   //limit switch depending
   IF IS_LINKED (di_LimitSwitchFwd) AND NOT IS_LINKED (di_LimitSwitchFwd2) THEN
      tmpFwd.pbDI := @di_LimitSwitchFwd;
   END_IF;
   IF IS_LINKED (di_LimitSwitchFwd2) THEN
      tmpFwd.pbDI := @di_LimitSwitchFwd2;
   END_IF;

   tmpBwd.pbDI := @di_LimitSwitchBwd;
   tmpBwd.pProfile := EMPTY;
   tmpFwd.pProfile := EMPTY;

ELSE
   //time depending
   tmpBwd.pbDI := EMPTY;
   tmpFwd.pbDI := EMPTY;
   tmpBwd.pProfile := EMPTY;
   tmpFwd.pProfile := EMPTY;

END_IF;

// update
sv_NozzleFwdMonData := tmpFwd;
sv_NozzleBwdMonData := tmpBwd;

;#END_EDIT_BLOCK END_ALGORITHM

POSTUPDATE_ALGORITHM pSetMovementMode ON PU_Task_3(1) WITH sv_NozzleMovementMode,sv_bInitStart

#BEGIN_EDIT_BLOCK
(**************************************** WARNING ********************************************
 *** The KEBA Kemro K2 System including software is not intended for safety control tasks! ***
 ***                       For further information see Comment tab!                        ***
 *********************************************************************************************)

//convert selector from HMI (position/time)
IF sv_NozzleMovementMode = nNozzleMovementModeTime THEN
   sv_MovementMode := nMoveTimeDependent;
ELSE
   //HMI selector = position
   IF IS_LINKED(ai_Position) THEN
      sv_MovementMode := nPositionDependent;
   ELSIF IS_LINKED(di_LimitSwitchFwd) THEN
      sv_MovementMode := nLimitSwitchDependent;
   ELSE
      //no tansducer or limit switch linked
      //(should not happen if project is created with AppCo)
      //-> set mode to time
      sv_MovementMode := nMoveTimeDependent;
   END_IF;
END_IF;

;#END_EDIT_BLOCK END_ALGORITHM

POSTUPDATE_ALGORITHM pFwdTimeReached ON PU_Task_3 WITH sv_bFwdTimeReached,sv_bInitStart

#BEGIN_EDIT_BLOCK
(**************************************** WARNING ********************************************
 *** The KEBA Kemro K2 System including software is not intended for safety control tasks! ***
 ***                       For further information see Comment tab!                        ***
 *********************************************************************************************)

IF sv_MovementMode = nMoveTimeDependent  THEN
   sv_bNozzleFwd := sv_bFwdTimeReached;
END_IF;

;#END_EDIT_BLOCK END_ALGORITHM

POSTUPDATE_ALGORITHM pBwdTimeReached ON PU_Task_3 WITH sv_bBwdTimeReached,sv_bInitStart

#BEGIN_EDIT_BLOCK
(**************************************** WARNING ********************************************
 *** The KEBA Kemro K2 System including software is not intended for safety control tasks! ***
 ***                       For further information see Comment tab!                        ***
 *********************************************************************************************)

IF sv_MovementMode <> nPositionDependent  THEN
   sv_bNozzleBwd := sv_bBwdTimeReached;
END_IF;

;#END_EDIT_BLOCK END_ALGORITHM

END_ALGORITHM_BLOCK

#END_OF_IEC_PART

@Puma @IecEditor 6 103 @Pou 25
@@@BEG_Comment@@@
@h    ! WARNING !
@h    The Kemro K2 system (including software) only meets category B according to EN 954-1,
@h    thus it is not intended for usage in safety-relevant control applications in the field
@h    of personal safety (e.g. emergency stop).
@h    To implement potentially necessary safety-relevant control tasks, always use additional
@h    external safety devices that are intended for the particular purpose, and meet the necessary
@h    functional safety.
@h    For further information see EN 954-1 (EN ISO 13849-1) and/or the K2-x00 user manual, chapter
@h    "CE conformity, directives and standards".

AB set the refernces for the endposition monitor blocks.
This refernces denpend on the selected movement mode (position, limit or time)
In time mode the endposition monitoring is also done by this block.
@@@END_Comment@@@

@BEG_Contents

@BEG_Func
@RT(17)FuncTreeContainer
3
@Var @RT(9)SET_ALARM @RT(0) @T @T @DERIVED 0 @F @RT(23)KEBA_STANDARD_PROCEDURE @F
@T
@BEG_Attrib
0 @RT(0) @RT(0)
@END_Attrib
1 1 @F @F @F @F

@Var @RT(23)START_PROCESS_ALGORITHM @RT(0) @T @T @DERIVED 0 @F @RT(23)KEBA_STANDARD_PROCEDURE @F
@T
@BEG_Attrib
0 @RT(0) @RT(0)
@END_Attrib
1 1 @F @F @F @F

@Var @RT(22)STOP_PROCESS_ALGORITHM @RT(0) @T @T @DERIVED 0 @F @RT(23)KEBA_STANDARD_PROCEDURE @F
@T
@BEG_Attrib
0 @RT(0) @RT(0)
@END_Attrib
1 1 @F @F @F @F

@END_Func

@BEG_Const
@RT(18)ConstTreeContainer
2
@Var @RT(18)nPositionDependent @RT(0) @T @T @DERIVED 0 @F @RT(14)tnMovementMode @F
@T
@BEG_Attrib
0 @RT(1)0 @RT(0)
@END_Attrib
1 1 @F @F @F @F

@Var @RT(18)nMoveTimeDependent @RT(0) @T @T @DERIVED 0 @F @RT(14)tnMovementMode @F
@T
@BEG_Attrib
0 @RT(1)2 @RT(0)
@END_Attrib
1 1 @F @F @F @F

@END_Const

@BEG_Export

@BEG_Kind
@ALGORITHM_BLOCK @RT(15)ABCheckSettings @STRUCTURED_TEXT
@RT(0) @RT(0) @RT(0)
@END_Kind

@BEG_Dcl
@RT(16)DclTreeContainer
16
@Var @RT(11)ai_Position @RT(0) @T @F @DT @RT(4)REAL @RT(0) @T @T @BASIC 0 @F
@F @F
@T
@BEG_Attrib
3 @RT(0) @RT(0) @RT(0)
@END_Attrib
1 8 @F @F @F @F

@Var @RT(15)sv_MovementMode @RT(0) @T @T @DERIVED 0 @T @T @DT @RT(14)tnMovementMode @RT(0) @T @T @UNKNOWN 0 @F
@F @F
@T
@BEG_Attrib
3 @RT(0) @RT(61)Nozzle Movement with Limitswitch or with position measurement @RT(0)
@END_Attrib
1 8 @F @F @F @F

@Var @RT(13)sv_bInitStart @RT(0) @T @F @DT @RT(4)BOOL @RT(0) @T @T @BASIC 0 @F
@F @F
@T
@BEG_Attrib
3 @RT(0) @RT(0) @RT(0)
@END_Attrib
1 8 @F @F @F @F

@Var @RT(19)sv_NozzleFwdMonData @RT(0) @T @T @DERIVED 0 @T @T @DT @RT(12)tsEndPosData @RT(0) @T @T @UNKNOWN 0 @F
@F @F
@T
@BEG_Attrib
3 @RT(0) @RT(0) @RT(0)
@END_Attrib
1 8 @F @F @F @F

@Var @RT(19)sv_NozzleBwdMonData @RT(0) @T @T @DERIVED 0 @T @T @DT @RT(12)tsEndPosData @RT(0) @T @T @UNKNOWN 0 @F
@F @F
@T
@BEG_Attrib
3 @RT(0) @RT(0) @RT(0)
@END_Attrib
1 8 @F @F @F @F

@Var @RT(17)di_LimitSwitchFwd @RT(0) @T @F @DT @RT(4)BOOL @RT(0) @T @T @BASIC 0 @F
@F @F
@T
@BEG_Attrib
3 @RT(0) @RT(0) @RT(0)
@END_Attrib
1 8 @F @F @F @F

@Var @RT(18)di_LimitSwitchFwd2 @RT(0) @T @F @DT @RT(4)BOOL @RT(0) @T @T @BASIC 0 @F
@F @F
@T
@BEG_Attrib
3 @RT(0) @RT(0) @RT(0)
@END_Attrib
1 8 @F @F @F @F

@Var @RT(9)PU_Task_3 @RT(0) @T @F @DT @RT(4)TASK @RT(0) @T @T @BASIC 0 @F
@F @F
@T
@BEG_Attrib
3 @RT(0) @RT(0) @RT(0)
@END_Attrib
1 7 @F @F @F @F

@Var @RT(19)sv_NozzleFwdProfVis @RT(0) @T @T @RENAMED 0 @T @T @DT @RT(16)KAPPL_VisProfile @RT(0) @T @T @UNKNOWN 0 @F
@F @F
@T
@BEG_Attrib
3 @RT(0) @RT(0) @RT(0)
@END_Attrib
1 8 @F @F @F @F

@Var @RT(19)sv_NozzleBwdProfVis @RT(0) @T @T @RENAMED 0 @T @T @DT @RT(16)KAPPL_VisProfile @RT(0) @T @T @UNKNOWN 0 @F
@F @F
@T
@BEG_Attrib
3 @RT(0) @RT(0) @RT(0)
@END_Attrib
1 8 @F @F @F @F

@Var @RT(17)di_LimitSwitchBwd @RT(0) @T @T @RENAMED 0 @T @T @DT @RT(4)BOOL @RT(0) @T @T @BASIC 0 @F
@F @F
@T
@BEG_Attrib
3 @RT(0) @RT(0) @RT(0)
@END_Attrib
1 8 @F @F @F @F

@Var @RT(13)sv_bNozzleFwd @RT(0) @T @F @DT @RT(4)BOOL @RT(0) @T @T @BASIC 0 @F
@F @F
@T
@BEG_Attrib
3 @RT(0) @RT(0) @RT(0)
@END_Attrib
1 8 @F @F @F @F

@Var @RT(13)sv_bNozzleBwd @RT(0) @T @F @DT @RT(4)BOOL @RT(0) @T @T @BASIC 0 @F
@F @F
@T
@BEG_Attrib
3 @RT(0) @RT(0) @RT(0)
@END_Attrib
1 8 @F @F @F @F

@Var @RT(18)sv_bFwdTimeReached @RT(0) @T @F @DT @RT(4)BOOL @RT(0) @T @T @BASIC 0 @F
@F @F
@T
@BEG_Attrib
3 @RT(0) @RT(110)nozzle fwd time reached (for time dependent nozzle control) (must be FastRetain: cyclical change in AutoCycle) @RT(0)
@END_Attrib
1 8 @F @F @F @F

@Var @RT(18)sv_bBwdTimeReached @RT(0) @T @F @DT @RT(4)BOOL @RT(0) @T @T @BASIC 0 @F
@F @F
@T
@BEG_Attrib
3 @RT(0) @RT(110)nozzle bwd time reached (for time dependent nozzle control) (must be FastRetain: cyclical change in AutoCycle) @RT(0)
@END_Attrib
1 8 @F @F @F @F

@Var @RT(21)sv_NozzleMovementMode @RT(0) @T @T @RENAMED 0 @T @T @DT @RT(20)tnNozzleMovementMode @RT(0) @T @T @UNKNOWN 0 @F
@F @F
@T
@BEG_Attrib
3 @RT(0) @RT(0) @RT(0)
@END_Attrib
1 8 @F @F @F @F

@END_Dcl

@END_Export

@BEG_Body

4

@BEG_Export

@BEG_Algo
@POSTUPDATE_ALGORITHM @RT(12)pModeChanged @STRUCTURED_TEXT
@RT(0) @RT(29)sv_MovementMode,sv_bInitStart @RT(9)PU_Task_3 @F @F
@END_Algo

@BEG_Dcl
@RT(16)DclTreeContainer
2
@Var @RT(6)tmpFwd @RT(0) @T @T @DERIVED 0 @T @T @DT @RT(12)tsEndPosData @RT(0) @T @T @UNKNOWN 0 @F
@F @F
@T
@BEG_Attrib
3 @RT(0) @RT(0) @RT(0)
@END_Attrib
1 4 @F @F @F @F

@Var @RT(6)tmpBwd @RT(0) @T @T @DERIVED 0 @T @T @DT @RT(12)tsEndPosData @RT(0) @T @T @UNKNOWN 0 @F
@F @F
@T
@BEG_Attrib
3 @RT(0) @RT(0) @RT(0)
@END_Attrib
1 4 @F @F @F @F

@END_Dcl

@END_Export

@BEG_Export

@BEG_Algo
@POSTUPDATE_ALGORITHM @RT(16)pSetMovementMode @STRUCTURED_TEXT
@RT(0) @RT(35)sv_NozzleMovementMode,sv_bInitStart @RT(12)PU_Task_3(1) @F @F
@END_Algo

@BEG_Dcl
@RT(16)DclTreeContainer
0
@END_Dcl

@END_Export

@BEG_Export

@BEG_Algo
@POSTUPDATE_ALGORITHM @RT(15)pFwdTimeReached @STRUCTURED_TEXT
@RT(0) @RT(32)sv_bFwdTimeReached,sv_bInitStart @RT(9)PU_Task_3 @F @F
@END_Algo

@BEG_Dcl
@RT(16)DclTreeContainer
0
@END_Dcl

@END_Export

@BEG_Export

@BEG_Algo
@POSTUPDATE_ALGORITHM @RT(15)pBwdTimeReached @STRUCTURED_TEXT
@RT(0) @RT(32)sv_bBwdTimeReached,sv_bInitStart @RT(9)PU_Task_3 @F @F
@END_Algo

@BEG_Dcl
@RT(16)DclTreeContainer
0
@END_Dcl

@END_Export

@BEG_Body
@TL(45)
(**************************************** WARNING ********************************************
 *** The KEBA Kemro K2 System including software is not intended for safety control tasks! ***
 ***                       For further information see Comment tab!                        ***
 *********************************************************************************************)

// update endposmon data when movement mode changes
// executed in PU_Task_3 so it is called before ABEndposMon.pParameterChanged

tmpFwd := sv_NozzleFwdMonData;
tmpBwd := sv_NozzleBwdMonData;

IF sv_MovementMode = nPositionDependent THEN
   //position depending
   tmpBwd.pbDI := EMPTY;
   tmpFwd.pbDI := EMPTY;
   tmpBwd.pProfile := @sv_NozzleBwdProfVis;
   tmpFwd.pProfile := @sv_NozzleFwdProfVis;

ELSIF sv_MovementMode = nLimitSwitchDependent THEN
   //limit switch depending
   IF IS_LINKED (di_LimitSwitchFwd) AND NOT IS_LINKED (di_LimitSwitchFwd2) THEN
      tmpFwd.pbDI := @di_LimitSwitchFwd;
   END_IF;
   IF IS_LINKED (di_LimitSwitchFwd2) THEN
      tmpFwd.pbDI := @di_LimitSwitchFwd2;
   END_IF;

   tmpBwd.pbDI := @di_LimitSwitchBwd;
   tmpBwd.pProfile := EMPTY;
   tmpFwd.pProfile := EMPTY;

ELSE
   //time depending
   tmpBwd.pbDI := EMPTY;
   tmpFwd.pbDI := EMPTY;
   tmpBwd.pProfile := EMPTY;
   tmpFwd.pProfile := EMPTY;

END_IF;

// update
sv_NozzleFwdMonData := tmpFwd;
sv_NozzleBwdMonData := tmpBwd;

@END_Body

@@@BEG_Comment@@@
@TL(0)

@@@END_Comment@@@

@BEG_Body
@TL(22)
(**************************************** WARNING ********************************************
 *** The KEBA Kemro K2 System including software is not intended for safety control tasks! ***
 ***                       For further information see Comment tab!                        ***
 *********************************************************************************************)

//convert selector from HMI (position/time)
IF sv_NozzleMovementMode = nNozzleMovementModeTime THEN
   sv_MovementMode := nMoveTimeDependent;
ELSE
   //HMI selector = position
   IF IS_LINKED(ai_Position) THEN
      sv_MovementMode := nPositionDependent;
   ELSIF IS_LINKED(di_LimitSwitchFwd) THEN
      sv_MovementMode := nLimitSwitchDependent;
   ELSE
      //no tansducer or limit switch linked
      //(should not happen if project is created with AppCo)
      //-> set mode to time
      sv_MovementMode := nMoveTimeDependent;
   END_IF;
END_IF;

@END_Body

@@@BEG_Comment@@@
@TL(0)

@@@END_Comment@@@

@BEG_Body
@TL(10)
(**************************************** WARNING ********************************************
 *** The KEBA Kemro K2 System including software is not intended for safety control tasks! ***
 ***                       For further information see Comment tab!                        ***
 *********************************************************************************************)

IF sv_MovementMode = nMoveTimeDependent  THEN
   sv_bNozzleFwd := sv_bFwdTimeReached;
END_IF;

@END_Body

@@@BEG_Comment@@@
@TL(0)

@@@END_Comment@@@

@BEG_Body
@TL(10)
(**************************************** WARNING ********************************************
 *** The KEBA Kemro K2 System including software is not intended for safety control tasks! ***
 ***                       For further information see Comment tab!                        ***
 *********************************************************************************************)

IF sv_MovementMode <> nPositionDependent  THEN
   sv_bNozzleBwd := sv_bBwdTimeReached;
END_IF;

@END_Body

@@@BEG_Comment@@@
@TL(0)

@@@END_Comment@@@
@END_Body

@END_Contents
